      "I847.0" { ExternalVisible := 'False'} : Bool := FALSE;   // I847.0
      "I847.1" { ExternalVisible := 'False'} : Bool := FALSE;   // I847.1
      "I847.2" { ExternalVisible := 'False'} : Bool := FALSE;   // I847.2
      "I847.3" { ExternalVisible := 'False'} : Bool := FALSE;   // I847.3
      "I847.4" { ExternalVisible := 'False'} : Bool := FALSE;   // I847.4
      "I847.5" { ExternalVisible := 'False'} : Bool := FALSE;   // I847.5
      "I847.6" { ExternalVisible := 'False'} : Bool := FALSE;   // I847.6
      "I847.7" { ExternalVisible := 'False'} : Bool := FALSE;   // I847.7
      "I848.0" { ExternalVisible := 'False'} : Bool := FALSE;   // I848.0
      "I848.1" { ExternalVisible := 'False'} : Bool := FALSE;   // I848.1
      "I848.2" { ExternalVisible := 'False'} : Bool := FALSE;   // I848.2
      "I848.3" { ExternalVisible := 'False'} : Bool := FALSE;   // I848.3
      "I848.4" { ExternalVisible := 'False'} : Bool := FALSE;   // I848.4
      "I848.5" { ExternalVisible := 'False'} : Bool := FALSE;   // I848.5
      "I848.6" { ExternalVisible := 'False'} : Bool := FALSE;   // I848.6
      "I848.7" { ExternalVisible := 'False'} : Bool := FALSE;   // I848.7
      "I849.0" { ExternalVisible := 'False'} : Bool := FALSE;   // I849.0
      "I849.1" { ExternalVisible := 'False'} : Bool := FALSE;   // I849.1
      "I849.2" { ExternalVisible := 'False'} : Bool := FALSE;   // I849.2
      "I849.3" { ExternalVisible := 'False'} : Bool := FALSE;   // I849.3
      "I849.4" { ExternalVisible := 'False'} : Bool := FALSE;   // I849.4
      "I849.5" { ExternalVisible := 'False'} : Bool := FALSE;   // I849.5
      "I849.6" { ExternalVisible := 'False'} : Bool := FALSE;   // I849.6
      "I849.7" { ExternalVisible := 'False'} : Bool := FALSE;   // I849.7
      "I850.0" { ExternalVisible := 'False'} : Bool := FALSE;   // I850.0
      "I850.1" { ExternalVisible := 'False'} : Bool := FALSE;   // I850.1
      "I850.2" { ExternalVisible := 'False'} : Bool := FALSE;   // I850.2
      "I850.3" { ExternalVisible := 'False'} : Bool := FALSE;   // I850.3
      "I850.4" { ExternalVisible := 'False'} : Bool := FALSE;   // I850.4
      "I850.5" { ExternalVisible := 'False'} : Bool := FALSE;   // I850.5
      "I850.6" { ExternalVisible := 'False'} : Bool := FALSE;   // I850.6
      "I850.7" { ExternalVisible := 'False'} : Bool := FALSE;   // I850.7
      "I851.0" { ExternalVisible := 'False'} : Bool := FALSE;   // I851.0
      "I851.1" { ExternalVisible := 'False'} : Bool := FALSE;   // I851.1
      "I851.2" { ExternalVisible := 'False'} : Bool := FALSE;   // I851.2
      "I851.3" { ExternalVisible := 'False'} : Bool := FALSE;   // I851.3
      "I851.4" { ExternalVisible := 'False'} : Bool := FALSE;   // I851.4
      "I851.5" { ExternalVisible := 'False'} : Bool := FALSE;   // I851.5
      "I851.6" { ExternalVisible := 'False'} : Bool := FALSE;   // I851.6
      "I851.7" { ExternalVisible := 'False'} : Bool := FALSE;   // I851.7
      "I852.0" { ExternalVisible := 'False'} : Bool := FALSE;   // I852.0
      "I852.1" { ExternalVisible := 'False'} : Bool := FALSE;   // I852.1
      "I852.2" { ExternalVisible := 'False'} : Bool := FALSE;   // I852.2
      "I852.3" { ExternalVisible := 'False'} : Bool := FALSE;   // I852.3
      "I852.4" { ExternalVisible := 'False'} : Bool := FALSE;   // I852.4
      "I852.5" { ExternalVisible := 'False'} : Bool := FALSE;   // I852.5
      "I852.6" { ExternalVisible := 'False'} : Bool := FALSE;   // I852.6
      "I852.7" { ExternalVisible := 'False'} : Bool := FALSE;   // I852.7
      "I853.0" { ExternalVisible := 'False'} : Bool := FALSE;   // I853.0
      "I853.1" { ExternalVisible := 'False'} : Bool := FALSE;   // I853.1
      "I853.2" { ExternalVisible := 'False'} : Bool := FALSE;   // I853.2
      "I853.3" { ExternalVisible := 'False'} : Bool := FALSE;   // I853.3
      "I853.4" { ExternalVisible := 'False'} : Bool := FALSE;   // I853.4
      "I853.5" { ExternalVisible := 'False'} : Bool := FALSE;   // I853.5
      "I853.6" { ExternalVisible := 'False'} : Bool := FALSE;   // I853.6
      "I853.7" { ExternalVisible := 'False'} : Bool := FALSE;   // I853.7
      "I854.0" { ExternalVisible := 'False'} : Bool := FALSE;   // I854.0
      "I854.1" { ExternalVisible := 'False'} : Bool := FALSE;   // I854.1
      "I854.2" { ExternalVisible := 'False'} : Bool := FALSE;   // I854.2
      "I854.3" { ExternalVisible := 'False'} : Bool := FALSE;   // I854.3
      "I854.4" { ExternalVisible := 'False'} : Bool := FALSE;   // I854.4
      "I854.5" { ExternalVisible := 'False'} : Bool := FALSE;   // I854.5
      "I854.6" { ExternalVisible := 'False'} : Bool := FALSE;   // I854.6
      "I854.7" { ExternalVisible := 'False'} : Bool := FALSE;   // I854.7
      "I855.0" { ExternalVisible := 'False'} : Bool := FALSE;   // I855.0
      "I855.1" { ExternalVisible := 'False'} : Bool := FALSE;   // I855.1
      "I855.2" { ExternalVisible := 'False'} : Bool := FALSE;   // I855.2
      "I855.3" { ExternalVisible := 'False'} : Bool := FALSE;   // I855.3
      "I855.4" { ExternalVisible := 'False'} : Bool := FALSE;   // I855.4
      "I855.5" { ExternalVisible := 'False'} : Bool := FALSE;   // I855.5
      "I855.6" { ExternalVisible := 'False'} : Bool := FALSE;   // I855.6
      "I855.7" { ExternalVisible := 'False'} : Bool := FALSE;   // I855.7
      "I856.0" { ExternalVisible := 'False'} : Bool := FALSE;   // I856.0
      "I856.1" { ExternalVisible := 'False'} : Bool := FALSE;   // I856.1
      "I856.2" { ExternalVisible := 'False'} : Bool := FALSE;   // I856.2
      "I856.3" { ExternalVisible := 'False'} : Bool := FALSE;   // I856.3
      "I856.4" { ExternalVisible := 'False'} : Bool := FALSE;   // I856.4
      "I856.5" { ExternalVisible := 'False'} : Bool := FALSE;   // I856.5
      "I856.6" { ExternalVisible := 'False'} : Bool := FALSE;   // I856.6
      "I856.7" { ExternalVisible := 'False'} : Bool := FALSE;   // I856.7
      "I857.0" { ExternalVisible := 'False'} : Bool := FALSE;   // I857.0
      "I857.1" { ExternalVisible := 'False'} : Bool := FALSE;   // I857.1
      "I857.2" { ExternalVisible := 'False'} : Bool := FALSE;   // I857.2
      "I857.3" { ExternalVisible := 'False'} : Bool := FALSE;   // I857.3
      "I857.4" { ExternalVisible := 'False'} : Bool := FALSE;   // I857.4
      "I857.5" { ExternalVisible := 'False'} : Bool := FALSE;   // I857.5
      "I857.6" { ExternalVisible := 'False'} : Bool := FALSE;   // I857.6
      "I857.7" { ExternalVisible := 'False'} : Bool := FALSE;   // I857.7
      "I858.0" { ExternalVisible := 'False'} : Bool := FALSE;   // I858.0
      "I858.1" { ExternalVisible := 'False'} : Bool := FALSE;   // I858.1
      "I858.2" { ExternalVisible := 'False'} : Bool := FALSE;   // I858.2
      "I858.3" { ExternalVisible := 'False'} : Bool := FALSE;   // I858.3
      "I858.4" { ExternalVisible := 'False'} : Bool := FALSE;   // I858.4
      "I858.5" { ExternalVisible := 'False'} : Bool := FALSE;   // I858.5
      "I858.6" { ExternalVisible := 'False'} : Bool := FALSE;   // I858.6
      "I858.7" { ExternalVisible := 'False'} : Bool := FALSE;   // I858.7
      "I859.0" { ExternalVisible := 'False'} : Bool := FALSE;   // I859.0
      "I859.1" { ExternalVisible := 'False'} : Bool := FALSE;   // I859.1
      "I859.2" { ExternalVisible := 'False'} : Bool := FALSE;   // I859.2
      "I859.3" { ExternalVisible := 'False'} : Bool := FALSE;   // I859.3
      "I859.4" { ExternalVisible := 'False'} : Bool := FALSE;   // I859.4
      "I859.5" { ExternalVisible := 'False'} : Bool := FALSE;   // I859.5
      "I859.6" { ExternalVisible := 'False'} : Bool := FALSE;   // I859.6
      "I859.7" { ExternalVisible := 'False'} : Bool := FALSE;   // I859.7
      "I860.0" { ExternalVisible := 'False'} : Bool := FALSE;   // I860.0
      "I860.1" { ExternalVisible := 'False'} : Bool := FALSE;   // I860.1
      "I860.2" { ExternalVisible := 'False'} : Bool := FALSE;   // I860.2
      "I860.3" { ExternalVisible := 'False'} : Bool := FALSE;   // I860.3
      "I860.4" { ExternalVisible := 'False'} : Bool := FALSE;   // I860.4
      "I860.5" { ExternalVisible := 'False'} : Bool := FALSE;   // I860.5
      "I860.6" { ExternalVisible := 'False'} : Bool := FALSE;   // I860.6
      "I860.7" { ExternalVisible := 'False'} : Bool := FALSE;   // I860.7
      "I861.0" { ExternalVisible := 'False'} : Bool := FALSE;   // I861.0
      "I861.1" { ExternalVisible := 'False'} : Bool := FALSE;   // I861.1
      "I861.2" { ExternalVisible := 'False'} : Bool := FALSE;   // I861.2
      "I861.3" { ExternalVisible := 'False'} : Bool := FALSE;   // I861.3
      "I861.4" { ExternalVisible := 'False'} : Bool := FALSE;   // I861.4
      "I861.5" { ExternalVisible := 'False'} : Bool := FALSE;   // I861.5
      "I861.6" { ExternalVisible := 'False'} : Bool := FALSE;   // I861.6
      "I861.7" { ExternalVisible := 'False'} : Bool := FALSE;   // I861.7
      "I862.0" { ExternalVisible := 'False'} : Bool := FALSE;   // I862.0
      "I862.1" { ExternalVisible := 'False'} : Bool := FALSE;   // I862.1
      "I862.2" { ExternalVisible := 'False'} : Bool := FALSE;   // I862.2
      "I862.3" { ExternalVisible := 'False'} : Bool := FALSE;   // I862.3
      "I862.4" { ExternalVisible := 'False'} : Bool := FALSE;   // I862.4
      "I862.5" { ExternalVisible := 'False'} : Bool := FALSE;   // I862.5
      "I862.6" { ExternalVisible := 'False'} : Bool := FALSE;   // I862.6
      "I862.7" { ExternalVisible := 'False'} : Bool := FALSE;   // I862.7
      "I863.0" { ExternalVisible := 'False'} : Bool := FALSE;   // I863.0
      "I863.1" { ExternalVisible := 'False'} : Bool := FALSE;   // I863.1
      "I863.2" { ExternalVisible := 'False'} : Bool := FALSE;   // I863.2
      "I863.3" { ExternalVisible := 'False'} : Bool := FALSE;   // I863.3
      "I863.4" { ExternalVisible := 'False'} : Bool := FALSE;   // I863.4
      "I863.5" { ExternalVisible := 'False'} : Bool := FALSE;   // I863.5
      "I863.6" { ExternalVisible := 'False'} : Bool := FALSE;   // I863.6
      "I863.7" { ExternalVisible := 'False'} : Bool := FALSE;   // I863.7
      "I864.0" { ExternalVisible := 'False'} : Bool := FALSE;   // I864.0
      "I864.1" { ExternalVisible := 'False'} : Bool := FALSE;   // I864.1
      "I864.2" { ExternalVisible := 'False'} : Bool := FALSE;   // I864.2
      "I864.3" { ExternalVisible := 'False'} : Bool := FALSE;   // I864.3
      "I864.4" { ExternalVisible := 'False'} : Bool := FALSE;   // I864.4
      "I864.5" { ExternalVisible := 'False'} : Bool := FALSE;   // I864.5
      "I864.6" { ExternalVisible := 'False'} : Bool := FALSE;   // I864.6
      "I864.7" { ExternalVisible := 'False'} : Bool := FALSE;   // I864.7
      "I865.0" { ExternalVisible := 'False'} : Bool := FALSE;   // I865.0
      "I865.1" { ExternalVisible := 'False'} : Bool := FALSE;   // I865.1
      "I865.2" { ExternalVisible := 'False'} : Bool := FALSE;   // I865.2
      "I865.3" { ExternalVisible := 'False'} : Bool := FALSE;   // I865.3
      "I865.4" { ExternalVisible := 'False'} : Bool := FALSE;   // I865.4
      "I865.5" { ExternalVisible := 'False'} : Bool := FALSE;   // I865.5
      "I865.6" { ExternalVisible := 'False'} : Bool := FALSE;   // I865.6
      "I865.7" { ExternalVisible := 'False'} : Bool := FALSE;   // I865.7
      "I866.0" { ExternalVisible := 'False'} : Bool := FALSE;   // I866.0
      "I866.1" { ExternalVisible := 'False'} : Bool := FALSE;   // I866.1
      "I866.2" { ExternalVisible := 'False'} : Bool := FALSE;   // I866.2
      "I866.3" { ExternalVisible := 'False'} : Bool := FALSE;   // I866.3
      "I866.4" { ExternalVisible := 'False'} : Bool := FALSE;   // I866.4
      "I866.5" { ExternalVisible := 'False'} : Bool := FALSE;   // I866.5
      "I866.6" { ExternalVisible := 'False'} : Bool := FALSE;   // I866.6
      "I866.7" { ExternalVisible := 'False'} : Bool := FALSE;   // I866.7
      "I867.0" { ExternalVisible := 'False'} : Bool := FALSE;   // I867.0
      "I867.1" { ExternalVisible := 'False'} : Bool := FALSE;   // I867.1
      "I867.2" { ExternalVisible := 'False'} : Bool := FALSE;   // I867.2
      "I867.3" { ExternalVisible := 'False'} : Bool := FALSE;   // I867.3
      "I867.4" { ExternalVisible := 'False'} : Bool := FALSE;   // I867.4
      "I867.5" { ExternalVisible := 'False'} : Bool := FALSE;   // I867.5
      "I867.6" { ExternalVisible := 'False'} : Bool := FALSE;   // I867.6
      "I867.7" { ExternalVisible := 'False'} : Bool := FALSE;   // I867.7
      "I868.0" { ExternalVisible := 'False'} : Bool := FALSE;   // I868.0
      "I868.1" { ExternalVisible := 'False'} : Bool := FALSE;   // I868.1
      "I868.2" { ExternalVisible := 'False'} : Bool := FALSE;   // I868.2
      "I868.3" { ExternalVisible := 'False'} : Bool := FALSE;   // I868.3
      "I868.4" { ExternalVisible := 'False'} : Bool := FALSE;   // I868.4
      "I868.5" { ExternalVisible := 'False'} : Bool := FALSE;   // I868.5
      "I868.6" { ExternalVisible := 'False'} : Bool := FALSE;   // I868.6
      "I868.7" { ExternalVisible := 'False'} : Bool := FALSE;   // I868.7
      "I869.0" { ExternalVisible := 'False'} : Bool := FALSE;   // I869.0
      "I869.1" { ExternalVisible := 'False'} : Bool := FALSE;   // I869.1
      "I869.2" { ExternalVisible := 'False'} : Bool := FALSE;   // I869.2
      "I869.3" { ExternalVisible := 'False'} : Bool := FALSE;   // I869.3
      "I869.4" { ExternalVisible := 'False'} : Bool := FALSE;   // I869.4
      "I869.5" { ExternalVisible := 'False'} : Bool := FALSE;   // I869.5
      "I869.6" { ExternalVisible := 'False'} : Bool := FALSE;   // I869.6
      "I869.7" { ExternalVisible := 'False'} : Bool := FALSE;   // I869.7
      "I870.0" { ExternalVisible := 'False'} : Bool := FALSE;   // I870.0
      "I870.1" { ExternalVisible := 'False'} : Bool := FALSE;   // I870.1
      "I870.2" { ExternalVisible := 'False'} : Bool := FALSE;   // I870.2
      "I870.3" { ExternalVisible := 'False'} : Bool := FALSE;   // I870.3
      "I870.4" { ExternalVisible := 'False'} : Bool := FALSE;   // I870.4
      "I870.5" { ExternalVisible := 'False'} : Bool := FALSE;   // I870.5
      "I870.6" { ExternalVisible := 'False'} : Bool := FALSE;   // I870.6
      "I870.7" { ExternalVisible := 'False'} : Bool := FALSE;   // I870.7
      "I871.0" { ExternalVisible := 'False'} : Bool := FALSE;   // I871.0
      "I871.1" { ExternalVisible := 'False'} : Bool := FALSE;   // I871.1
      "I871.2" { ExternalVisible := 'False'} : Bool := FALSE;   // I871.2
      "I871.3" { ExternalVisible := 'False'} : Bool := FALSE;   // I871.3
      "I871.4" { ExternalVisible := 'False'} : Bool := FALSE;   // I871.4
      "I871.5" { ExternalVisible := 'False'} : Bool := FALSE;   // I871.5
      "I871.6" { ExternalVisible := 'False'} : Bool := FALSE;   // I871.6
      "I871.7" { ExternalVisible := 'False'} : Bool := FALSE;   // I871.7
      "I872.0" { ExternalVisible := 'False'} : Bool := FALSE;   // I872.0
      "I872.1" { ExternalVisible := 'False'} : Bool := FALSE;   // I872.1
      "I872.2" { ExternalVisible := 'False'} : Bool := FALSE;   // I872.2
      "I872.3" { ExternalVisible := 'False'} : Bool := FALSE;   // I872.3
      "I872.4" { ExternalVisible := 'False'} : Bool := FALSE;   // I872.4
      "I872.5" { ExternalVisible := 'False'} : Bool := FALSE;   // I872.5
      "I872.6" { ExternalVisible := 'False'} : Bool := FALSE;   // I872.6
      "I872.7" { ExternalVisible := 'False'} : Bool := FALSE;   // I872.7
      "I873.0" { ExternalVisible := 'False'} : Bool := FALSE;   // I873.0
      "I873.1" { ExternalVisible := 'False'} : Bool := FALSE;   // I873.1
      "I873.2" { ExternalVisible := 'False'} : Bool := FALSE;   // I873.2
      "I873.3" { ExternalVisible := 'False'} : Bool := FALSE;   // I873.3
      "I873.4" { ExternalVisible := 'False'} : Bool := FALSE;   // I873.4
      "I873.5" { ExternalVisible := 'False'} : Bool := FALSE;   // I873.5
      "I873.6" { ExternalVisible := 'False'} : Bool := FALSE;   // I873.6
      "I873.7" { ExternalVisible := 'False'} : Bool := FALSE;   // I873.7
      "I874.0" { ExternalVisible := 'False'} : Bool := FALSE;   // I874.0
      "I874.1" { ExternalVisible := 'False'} : Bool := FALSE;   // I874.1
      "I874.2" { ExternalVisible := 'False'} : Bool := FALSE;   // I874.2
      "I874.3" { ExternalVisible := 'False'} : Bool := FALSE;   // I874.3
      "I874.4" { ExternalVisible := 'False'} : Bool := FALSE;   // I874.4
      "I874.5" { ExternalVisible := 'False'} : Bool := FALSE;   // I874.5
      "I874.6" { ExternalVisible := 'False'} : Bool := FALSE;   // I874.6
      "I874.7" { ExternalVisible := 'False'} : Bool := FALSE;   // I874.7
      "I875.0" { ExternalVisible := 'False'} : Bool := FALSE;   // I875.0
      "I875.1" { ExternalVisible := 'False'} : Bool := FALSE;   // I875.1
      "I875.2" { ExternalVisible := 'False'} : Bool := FALSE;   // I875.2
      "I875.3" { ExternalVisible := 'False'} : Bool := FALSE;   // I875.3
      "I875.4" { ExternalVisible := 'False'} : Bool := FALSE;   // I875.4
      "I875.5" { ExternalVisible := 'False'} : Bool := FALSE;   // I875.5
      "I875.6" { ExternalVisible := 'False'} : Bool := FALSE;   // I875.6
      "I875.7" { ExternalVisible := 'False'} : Bool := FALSE;   // I875.7
      "I876.0" { ExternalVisible := 'False'} : Bool := FALSE;   // I876.0
      "I876.1" { ExternalVisible := 'False'} : Bool := FALSE;   // I876.1
      "I876.2" { ExternalVisible := 'False'} : Bool := FALSE;   // I876.2
      "I876.3" { ExternalVisible := 'False'} : Bool := FALSE;   // I876.3
      "I876.4" { ExternalVisible := 'False'} : Bool := FALSE;   // I876.4
      "I876.5" { ExternalVisible := 'False'} : Bool := FALSE;   // I876.5
      "I876.6" { ExternalVisible := 'False'} : Bool := FALSE;   // I876.6
      "I876.7" { ExternalVisible := 'False'} : Bool := FALSE;   // I876.7
      "I877.0" { ExternalVisible := 'False'} : Bool := FALSE;   // I877.0
      "I877.1" { ExternalVisible := 'False'} : Bool := FALSE;   // I877.1
      "I877.2" { ExternalVisible := 'False'} : Bool := FALSE;   // I877.2
      "I877.3" { ExternalVisible := 'False'} : Bool := FALSE;   // I877.3
      "I877.4" { ExternalVisible := 'False'} : Bool := FALSE;   // I877.4
      "I877.5" { ExternalVisible := 'False'} : Bool := FALSE;   // I877.5
      "I877.6" { ExternalVisible := 'False'} : Bool := FALSE;   // I877.6
      "I877.7" { ExternalVisible := 'False'} : Bool := FALSE;   // I877.7
      "I878.0" { ExternalVisible := 'False'} : Bool := FALSE;   // I878.0
      "I878.1" { ExternalVisible := 'False'} : Bool := FALSE;   // I878.1
      "I878.2" { ExternalVisible := 'False'} : Bool := FALSE;   // I878.2
      "I878.3" { ExternalVisible := 'False'} : Bool := FALSE;   // I878.3
      "I878.4" { ExternalVisible := 'False'} : Bool := FALSE;   // I878.4
      "I878.5" { ExternalVisible := 'False'} : Bool := FALSE;   // I878.5
      "I878.6" { ExternalVisible := 'False'} : Bool := FALSE;   // I878.6
      "I878.7" { ExternalVisible := 'False'} : Bool := FALSE;   // I878.7
      "I879.0" { ExternalVisible := 'False'} : Bool := FALSE;   // I879.0
      "I879.1" { ExternalVisible := 'False'} : Bool := FALSE;   // I879.1
      "I879.2" { ExternalVisible := 'False'} : Bool := FALSE;   // I879.2
      "I879.3" { ExternalVisible := 'False'} : Bool := FALSE;   // I879.3
      "I879.4" { ExternalVisible := 'False'} : Bool := FALSE;   // I879.4
      "I879.5" { ExternalVisible := 'False'} : Bool := FALSE;   // I879.5
      "I879.6" { ExternalVisible := 'False'} : Bool := FALSE;   // I879.6
      "I879.7" { ExternalVisible := 'False'} : Bool := FALSE;   // I879.7
      "I880.0" { ExternalVisible := 'False'} : Bool := FALSE;   // I880.0
      "I880.1" { ExternalVisible := 'False'} : Bool := FALSE;   // I880.1
      "I880.2" { ExternalVisible := 'False'} : Bool := FALSE;   // I880.2
      "I880.3" { ExternalVisible := 'False'} : Bool := FALSE;   // I880.3
      "I880.4" { ExternalVisible := 'False'} : Bool := FALSE;   // I880.4
      "I880.5" { ExternalVisible := 'False'} : Bool := FALSE;   // I880.5
      "I880.6" { ExternalVisible := 'False'} : Bool := FALSE;   // I880.6
      "I880.7" { ExternalVisible := 'False'} : Bool := FALSE;   // I880.7
      "I881.0" { ExternalVisible := 'False'} : Bool := FALSE;   // I881.0
      "I881.1" { ExternalVisible := 'False'} : Bool := FALSE;   // I881.1
      "I881.2" { ExternalVisible := 'False'} : Bool := FALSE;   // I881.2
      "I881.3" { ExternalVisible := 'False'} : Bool := FALSE;   // I881.3
      "I881.4" { ExternalVisible := 'False'} : Bool := FALSE;   // I881.4
      "I881.5" { ExternalVisible := 'False'} : Bool := FALSE;   // I881.5
      "I881.6" { ExternalVisible := 'False'} : Bool := FALSE;   // I881.6
      "I881.7" { ExternalVisible := 'False'} : Bool := FALSE;   // I881.7
      "I882.0" { ExternalVisible := 'False'} : Bool := FALSE;   // I882.0
      "I882.1" { ExternalVisible := 'False'} : Bool := FALSE;   // I882.1
      "I882.2" { ExternalVisible := 'False'} : Bool := FALSE;   // I882.2
      "I882.3" { ExternalVisible := 'False'} : Bool := FALSE;   // I882.3
      "I882.4" { ExternalVisible := 'False'} : Bool := FALSE;   // I882.4
      "I882.5" { ExternalVisible := 'False'} : Bool := FALSE;   // I882.5
      "I882.6" { ExternalVisible := 'False'} : Bool := FALSE;   // I882.6
      "I882.7" { ExternalVisible := 'False'} : Bool := FALSE;   // I882.7
      "I883.0" { ExternalVisible := 'False'} : Bool := FALSE;   // I883.0
      "I883.1" { ExternalVisible := 'False'} : Bool := FALSE;   // I883.1
      "I883.2" { ExternalVisible := 'False'} : Bool := FALSE;   // I883.2
      "I883.3" { ExternalVisible := 'False'} : Bool := FALSE;   // I883.3
      "I883.4" { ExternalVisible := 'False'} : Bool := FALSE;   // I883.4
      "I883.5" { ExternalVisible := 'False'} : Bool := FALSE;   // I883.5
      "I883.6" { ExternalVisible := 'False'} : Bool := FALSE;   // I883.6
      "I883.7" { ExternalVisible := 'False'} : Bool := FALSE;   // I883.7
      "I884.0" { ExternalVisible := 'False'} : Bool := FALSE;   // I884.0
      "I884.1" { ExternalVisible := 'False'} : Bool := FALSE;   // I884.1
      "I884.2" { ExternalVisible := 'False'} : Bool := FALSE;   // I884.2
      "I884.3" { ExternalVisible := 'False'} : Bool := FALSE;   // I884.3
      "I884.4" { ExternalVisible := 'False'} : Bool := FALSE;   // I884.4
      "I884.5" { ExternalVisible := 'False'} : Bool := FALSE;   // I884.5
      "I884.6" { ExternalVisible := 'False'} : Bool := FALSE;   // I884.6
      "I884.7" { ExternalVisible := 'False'} : Bool := FALSE;   // I884.7
      "I885.0" { ExternalVisible := 'False'} : Bool := FALSE;   // I885.0
      "I885.1" { ExternalVisible := 'False'} : Bool := FALSE;   // I885.1
      "I885.2" { ExternalVisible := 'False'} : Bool := FALSE;   // I885.2
      "I885.3" { ExternalVisible := 'False'} : Bool := FALSE;   // I885.3
      "I885.4" { ExternalVisible := 'False'} : Bool := FALSE;   // I885.4
      "I885.5" { ExternalVisible := 'False'} : Bool := FALSE;   // I885.5
      "I885.6" { ExternalVisible := 'False'} : Bool := FALSE;   // I885.6
      "I885.7" { ExternalVisible := 'False'} : Bool := FALSE;   // I885.7
      "I886.0" { ExternalVisible := 'False'} : Bool := FALSE;   // I886.0
      "I886.1" { ExternalVisible := 'False'} : Bool := FALSE;   // I886.1
      "I886.2" { ExternalVisible := 'False'} : Bool := FALSE;   // I886.2
      "I886.3" { ExternalVisible := 'False'} : Bool := FALSE;   // I886.3
      "I886.4" { ExternalVisible := 'False'} : Bool := FALSE;   // I886.4
      "I886.5" { ExternalVisible := 'False'} : Bool := FALSE;   // I886.5
      "I886.6" { ExternalVisible := 'False'} : Bool := FALSE;   // I886.6
      "I886.7" { ExternalVisible := 'False'} : Bool := FALSE;   // I886.7
      "I887.0" { ExternalVisible := 'False'} : Bool := FALSE;   // I887.0
      "I887.1" { ExternalVisible := 'False'} : Bool := FALSE;   // I887.1
      "I887.2" { ExternalVisible := 'False'} : Bool := FALSE;   // I887.2
      "I887.3" { ExternalVisible := 'False'} : Bool := FALSE;   // I887.3
      "I887.4" { ExternalVisible := 'False'} : Bool := FALSE;   // I887.4
      "I887.5" { ExternalVisible := 'False'} : Bool := FALSE;   // I887.5
      "I887.6" { ExternalVisible := 'False'} : Bool := FALSE;   // I887.6
      "I887.7" { ExternalVisible := 'False'} : Bool := FALSE;   // I887.7
      "I888.0" { ExternalVisible := 'False'} : Bool := FALSE;   // I888.0
      "I888.1" { ExternalVisible := 'False'} : Bool := FALSE;   // I888.1
      "I888.2" { ExternalVisible := 'False'} : Bool := FALSE;   // I888.2
      "I888.3" { ExternalVisible := 'False'} : Bool := FALSE;   // I888.3
      "I888.4" { ExternalVisible := 'False'} : Bool := FALSE;   // I888.4
      "I888.5" { ExternalVisible := 'False'} : Bool := FALSE;   // I888.5
      "I888.6" { ExternalVisible := 'False'} : Bool := FALSE;   // I888.6
      "I888.7" { ExternalVisible := 'False'} : Bool := FALSE;   // I888.7
      "I889.0" { ExternalVisible := 'False'} : Bool := FALSE;   // I889.0
      "I889.1" { ExternalVisible := 'False'} : Bool := FALSE;   // I889.1
      "I889.2" { ExternalVisible := 'False'} : Bool := FALSE;   // I889.2
      "I889.3" { ExternalVisible := 'False'} : Bool := FALSE;   // I889.3
      "I889.4" { ExternalVisible := 'False'} : Bool := FALSE;   // I889.4
      "I889.5" { ExternalVisible := 'False'} : Bool := FALSE;   // I889.5
      "I889.6" { ExternalVisible := 'False'} : Bool := FALSE;   // I889.6
      "I889.7" { ExternalVisible := 'False'} : Bool := FALSE;   // I889.7
      "I890.0" { ExternalVisible := 'False'} : Bool := FALSE;   // I890.0
      "I890.1" { ExternalVisible := 'False'} : Bool := FALSE;   // I890.1
      "I890.2" { ExternalVisible := 'False'} : Bool := FALSE;   // I890.2
      "I890.3" { ExternalVisible := 'False'} : Bool := FALSE;   // I890.3
      "I890.4" { ExternalVisible := 'False'} : Bool := FALSE;   // I890.4
      "I890.5" { ExternalVisible := 'False'} : Bool := FALSE;   // I890.5
      "I890.6" { ExternalVisible := 'False'} : Bool := FALSE;   // I890.6
      "I890.7" { ExternalVisible := 'False'} : Bool := FALSE;   // I890.7
      "I891.0" { ExternalVisible := 'False'} : Bool := FALSE;   // I891.0
      "I891.1" { ExternalVisible := 'False'} : Bool := FALSE;   // I891.1
      "I891.2" { ExternalVisible := 'False'} : Bool := FALSE;   // I891.2
      "I891.3" { ExternalVisible := 'False'} : Bool := FALSE;   // I891.3
      "I891.4" { ExternalVisible := 'False'} : Bool := FALSE;   // I891.4
      "I891.5" { ExternalVisible := 'False'} : Bool := FALSE;   // I891.5
      "I891.6" { ExternalVisible := 'False'} : Bool := FALSE;   // I891.6
      "I891.7" { ExternalVisible := 'False'} : Bool := FALSE;   // I891.7
      "I892.0" { ExternalVisible := 'False'} : Bool := FALSE;   // I892.0
      "I892.1" { ExternalVisible := 'False'} : Bool := FALSE;   // I892.1
      "I892.2" { ExternalVisible := 'False'} : Bool := FALSE;   // I892.2
      "I892.3" { ExternalVisible := 'False'} : Bool := FALSE;   // I892.3
      "I892.4" { ExternalVisible := 'False'} : Bool := FALSE;   // I892.4
      "I892.5" { ExternalVisible := 'False'} : Bool := FALSE;   // I892.5
      "I892.6" { ExternalVisible := 'False'} : Bool := FALSE;   // I892.6
      "I892.7" { ExternalVisible := 'False'} : Bool := FALSE;   // I892.7
      "I893.0" { ExternalVisible := 'False'} : Bool := FALSE;   // I893.0
      "I893.1" { ExternalVisible := 'False'} : Bool := FALSE;   // I893.1
      "I893.2" { ExternalVisible := 'False'} : Bool := FALSE;   // I893.2
      "I893.3" { ExternalVisible := 'False'} : Bool := FALSE;   // I893.3
      "I893.4" { ExternalVisible := 'False'} : Bool := FALSE;   // I893.4
      "I893.5" { ExternalVisible := 'False'} : Bool := FALSE;   // I893.5
      "I893.6" { ExternalVisible := 'False'} : Bool := FALSE;   // I893.6
      "I893.7" { ExternalVisible := 'False'} : Bool := FALSE;   // I893.7
      "I894.0" { ExternalVisible := 'False'} : Bool := FALSE;   // I894.0
      "I894.1" { ExternalVisible := 'False'} : Bool := FALSE;   // I894.1
      "I894.2" { ExternalVisible := 'False'} : Bool := FALSE;   // I894.2
      "I894.3" { ExternalVisible := 'False'} : Bool := FALSE;   // I894.3
      "I894.4" { ExternalVisible := 'False'} : Bool := FALSE;   // I894.4
      "I894.5" { ExternalVisible := 'False'} : Bool := FALSE;   // I894.5
      "I894.6" { ExternalVisible := 'False'} : Bool := FALSE;   // I894.6
      "I894.7" { ExternalVisible := 'False'} : Bool := FALSE;   // I894.7
      "I895.0" { ExternalVisible := 'False'} : Bool := FALSE;   // I895.0
      "I895.1" { ExternalVisible := 'False'} : Bool := FALSE;   // I895.1
      "I895.2" { ExternalVisible := 'False'} : Bool := FALSE;   // I895.2
      "I895.3" { ExternalVisible := 'False'} : Bool := FALSE;   // I895.3
      "I895.4" { ExternalVisible := 'False'} : Bool := FALSE;   // I895.4
      "I895.5" { ExternalVisible := 'False'} : Bool := FALSE;   // I895.5
      "I895.6" { ExternalVisible := 'False'} : Bool := FALSE;   // I895.6
      "I895.7" { ExternalVisible := 'False'} : Bool := FALSE;   // I895.7
      "I896.0" { ExternalVisible := 'False'} : Bool := FALSE;   // I896.0
      "I896.1" { ExternalVisible := 'False'} : Bool := FALSE;   // I896.1
      "I896.2" { ExternalVisible := 'False'} : Bool := FALSE;   // I896.2
      "I896.3" { ExternalVisible := 'False'} : Bool := FALSE;   // I896.3
      "I896.4" { ExternalVisible := 'False'} : Bool := FALSE;   // I896.4
      "I896.5" { ExternalVisible := 'False'} : Bool := FALSE;   // I896.5
      "I896.6" { ExternalVisible := 'False'} : Bool := FALSE;   // I896.6
      "I896.7" { ExternalVisible := 'False'} : Bool := FALSE;   // I896.7
      "I897.0" { ExternalVisible := 'False'} : Bool := FALSE;   // I897.0
      "I897.1" { ExternalVisible := 'False'} : Bool := FALSE;   // I897.1
      "I897.2" { ExternalVisible := 'False'} : Bool := FALSE;   // I897.2
      "I897.3" { ExternalVisible := 'False'} : Bool := FALSE;   // I897.3
      "I897.4" { ExternalVisible := 'False'} : Bool := FALSE;   // I897.4
      "I897.5" { ExternalVisible := 'False'} : Bool := FALSE;   // I897.5
      "I897.6" { ExternalVisible := 'False'} : Bool := FALSE;   // I897.6
      "I897.7" { ExternalVisible := 'False'} : Bool := FALSE;   // I897.7
      "I898.0" { ExternalVisible := 'False'} : Bool := FALSE;   // I898.0
      "I898.1" { ExternalVisible := 'False'} : Bool := FALSE;   // I898.1
      "I898.2" { ExternalVisible := 'False'} : Bool := FALSE;   // I898.2
      "I898.3" { ExternalVisible := 'False'} : Bool := FALSE;   // I898.3
      "I898.4" { ExternalVisible := 'False'} : Bool := FALSE;   // I898.4
      "I898.5" { ExternalVisible := 'False'} : Bool := FALSE;   // I898.5
      "I898.6" { ExternalVisible := 'False'} : Bool := FALSE;   // I898.6
      "I898.7" { ExternalVisible := 'False'} : Bool := FALSE;   // I898.7
      "I899.0" { ExternalVisible := 'False'} : Bool := FALSE;   // I899.0
      "I899.1" { ExternalVisible := 'False'} : Bool := FALSE;   // I899.1
      "I899.2" { ExternalVisible := 'False'} : Bool := FALSE;   // I899.2
      "I899.3" { ExternalVisible := 'False'} : Bool := FALSE;   // I899.3
      "I899.4" { ExternalVisible := 'False'} : Bool := FALSE;   // I899.4
      "I899.5" { ExternalVisible := 'False'} : Bool := FALSE;   // I899.5
      "I899.6" { ExternalVisible := 'False'} : Bool := FALSE;   // I899.6
      "I899.7" { ExternalVisible := 'False'} : Bool := FALSE;   // I899.7
      "I900.0" { ExternalVisible := 'False'} : Bool := FALSE;   // I900.0
      "I900.1" { ExternalVisible := 'False'} : Bool := FALSE;   // I900.1
      "I900.2" { ExternalVisible := 'False'} : Bool := FALSE;   // I900.2
      "I900.3" { ExternalVisible := 'False'} : Bool := FALSE;   // I900.3
      "I900.4" { ExternalVisible := 'False'} : Bool := FALSE;   // I900.4
      "I900.5" { ExternalVisible := 'False'} : Bool := FALSE;   // I900.5
      "I900.6" { ExternalVisible := 'False'} : Bool := FALSE;   // I900.6
      "I900.7" { ExternalVisible := 'False'} : Bool := FALSE;   // I900.7
   END_VAR
BEGIN
END_DATA_BLOCK
